INTERFACE I_Halt

PROPERTY ExecHalt : BOOL
SET
END_SET
END_PROPERTY

METHOD Halt
VAR_INPUT
	Execute : BOOL;
    Deceleration : LREAL := 0.0;
    Jerk : LREAL := 0.0;
    BufferMode	: MC_BufferMode := MC_BufferMode.MC_Aborting;
END_VAR
END_METHOD

PROPERTY HaltActive : BOOL
GET
END_GET
END_PROPERTY

PROPERTY HaltBufferMode : MC_BufferMode
SET
END_SET
END_PROPERTY

PROPERTY HaltBusy : BOOL
GET
END_GET
END_PROPERTY

PROPERTY HaltDeceleration : LREAL
SET
END_SET
END_PROPERTY

PROPERTY HaltDone : BOOL
GET
END_GET
END_PROPERTY

PROPERTY HaltError : BOOL
GET
END_GET
END_PROPERTY

PROPERTY HaltErrorID : UDINT
GET
END_GET
END_PROPERTY

PROPERTY HaltJerk : LREAL
SET
END_SET
END_PROPERTY

END_INTERFACE

(* stored: Version 1.1.0.1
   Itf I_Halt: Id {14029942-f501-4700-ae44-ffd198ee0804}
   Property ExecHalt: Id {9b612b02-e6fe-499a-8b3e-79abf4f94e66}
   Set Set: Id {e554b9d8-8fe8-459e-8090-74311562fc7b}
   Method Halt: Id {d4ac7148-c266-4f03-80ec-1cc697d63c31}
   Property HaltActive: Id {931a7ba1-a94e-4370-afcb-3d6e40f3a0e7}
   Get Get: Id {2f305331-f614-4dee-9034-de312cec5ae6}
   Property HaltBufferMode: Id {c603523d-3e6d-406a-9c28-c785372ac4f9}
   Set Set: Id {588c8203-51c6-4070-a58c-c342e4c0f7ed}
   Property HaltBusy: Id {8ae225ed-f5ab-4332-acdc-c3e42aaded5a}
   Get Get: Id {3e6dd916-c2f0-4863-b925-df304bd91ced}
   Property HaltDeceleration: Id {b0d9bc59-f323-45f2-ad94-a6d3058ecc72}
   Set Set: Id {966d937b-e477-4fec-8d56-cf82ad9e7bae}
   Property HaltDone: Id {8055714d-6e20-4cf5-91fc-9c7794dae23b}
   Get Get: Id {092a4d2a-b995-4f67-bc71-fed54ee1f3b0}
   Property HaltError: Id {b9ba3ac4-f6e9-478b-a790-070b8eee962a}
   Get Get: Id {8e5fdeaf-b675-4a22-8ff0-52fbc36f0b62}
   Property HaltErrorID: Id {a7865411-559f-48f8-ae61-133b29ccf9ba}
   Get Get: Id {00fd4576-9142-4e39-a11d-09bd0f063a59}
   Property HaltJerk: Id {9732ff75-ccee-491e-a82e-79d01f721a28}
   Set Set: Id {41efdf2e-48ec-4a96-82ff-f2904126f038} *)
